{attribute 'GeneratedUsingTerminal: EK1122-0000-0018'}
{attribute addProperty BoxType "EK1122-0000-0018"}
{attribute addProperty Id "Beckhoff_EM7xxxsub_EK1100EK1100_1FC0878B2"}
{attribute addProperty CRC "3739850570"}
{attribute addProperty Size "2"}
TYPE Beckhoff_EM7xxxEK1122_DEE9974A EXTENDS EK1122_1FC0878B :
STRUCT
	{attribute addProperty Name "Beckhoff_EM7xxxsub_EK1100"}
	{attribute addProperty PreviousPort "Beckhoff EM7xxxEK1122 : D"}
	Beckhoff_EM7xxxsub_EK1100 : EK1100_1FC0878B;
END_STRUCT
END_TYPE

(* stored: Version 1.2.0.0, ProductVersion 3.1.4024.9
   DUT Beckhoff_EM7xxxEK1122_DEE9974A: Id {9f0762fe-834c-482b-814f-bb461c1ec117} *)
